PROGRAM P_Demo_FB_HVACCmdCtrlSystem1Stage
VAR
    fb : FB_HVACCmdCtrlSystem1Stage;                            // 被演示 FB 实例
    eDataSecurityType_in : E_HVACDataSecurityType ;
    bSetDefault_in : BOOL := FALSE;
    bEnable_in : BOOL := FALSE;
    eCtrlModeActuator_in : E_HVACActuatorMode ;
    bExternalRequest_in : BOOL := FALSE;
    bTimeScheduler_in : BOOL := FALSE;
    bReset_in : BOOL := FALSE;
    ePlantMode_io : E_HVACPlantMode ;
    eExternalRequestMode_io : E_HVACExternalRequestMode ;
    tOffDelay_io : TIME := T#0S;
    bOn_out : BOOL;
    eStateModeActuator_out : E_HVACActuatorMode;
    bRequestScheduler_out : BOOL;
    bRequestExternal_out : BOOL;
    bInvalidParameter_out : BOOL;
END_VAR

// ============================================================================
// Tc2_HVAC.FB_HVACCmdCtrlSystem1Stage 演示程序
// ============================================================================
// 场景：把本 FB 实例化到一个 PLC 程序里，每周期单次调用；按需要把 VAR_INPUT 与
//       VAR_IN_OUT 接到工程信号；VAR_OUTPUT 写入对应监视变量。
// 价值：使用本 FB 比手写状态机 / 控制算法节省大量代码；与 Tc2_HVAC 体系内其它 FB
//       直接对接，命名 / 持久化 / 模式仲裁等约定一致。具体语义见 FB_HVACCmdCtrlSystem1Stage.md 主文档。
// 验证步骤：
//   1. 右键 PLC 项目下 POUs 文件夹 → Add → Existing Item → 选本 .TcPOU 文件
//   2. 引用 Tc2_HVAC（References → Add library）
//   3. 编译 → 登录 → 运行
//   4. 在线写各 *_in 输入信号触发 FB；在线 monitor *_out 引脚观察状态
// ============================================================================

fb(
    eDataSecurityType := eDataSecurityType_in,
    bSetDefault := bSetDefault_in,
    bEnable := bEnable_in,
    eCtrlModeActuator := eCtrlModeActuator_in,
    bExternalRequest := bExternalRequest_in,
    bTimeScheduler := bTimeScheduler_in,
    bReset := bReset_in,
    ePlantMode := ePlantMode_io,
    eExternalRequestMode := eExternalRequestMode_io,
    tOffDelay := tOffDelay_io,
    bOn => bOn_out,
    eStateModeActuator => eStateModeActuator_out,
    bRequestScheduler => bRequestScheduler_out,
    bRequestExternal => bRequestExternal_out,
    bInvalidParameter => bInvalidParameter_out
);

END_PROGRAM

(* stored: Version 1.1.0.1, ProductVersion 3.1.4024.5
   POU P_Demo_FB_HVACCmdCtrlSystem1Stage: Id {3de059b2-fb03-5795-96ac-46c6bcdeb467}, SpecialFunc None *)
